Omron CX-Programmer project NewProject (CX-Programmer 9.61)

# PLC NewPLC1: CP1E N30

## Global symbols (name address type ; comment)
0.00 BOOL  ; PB2
0.01 BOOL  ; PB3
100.00 BOOL  ; lampu
T000 BOOL  ; Timer 1

## Program NewProgram1 (cyclic task 0)

### Section Section1

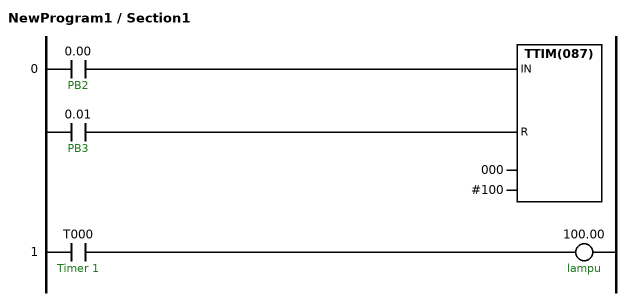
; rung 0
LD 0.00  ; PB2
LD 0.01  ; PB3
TTIM(087) 000 #100  ; Timer 1
; rung 1
LD T000  ; Timer 1
OUT 100.00  ; lampu

### Section END
; rung 0
END(001)